FUNCTION_BLOCK FB_RunClock
// LREAL: Long Real decimal number	
// BOOL: True/False

// Input variables
VAR_INPUT
	bStart 		: BOOL; 		// Set to true
	bStop 		: BOOL; 		// Stop button on controller
	fCycleTime  : LREAL; 		// Time step [s]
END_VAR

// Output variables
VAR_OUTPUT
	fTime : LREAL; 		// Output (time)
END_VAR

// Variables
VAR
	bOnOff : BOOL; 		// True/False
END_VAR

IF bStop OR (G_Work.eStatus = E_Status.Off) THEN 	// If stop button is pressed or system is off 
	bOnOff := FALSE; 
	fTime := 0.0; 
ELSIF bOnOff OR bStart THEN 	// If system is online/start button pushed, start timer
	bOnOff := TRUE;
	fTime := fTime + fCycleTime;
END_IF

END_FUNCTION_BLOCK

(* stored: Version 1.1.0.1
   POU FB_RunClock: Id {72885421-59e1-4582-bbdc-64c324631609}, SpecialFunc None *)
